{attribute 'GeneratedUsingTerminal: EP3356-0022-0016'}
{attribute addProperty BoxType "EP3356-0022-0016"}
{attribute addProperty Id "CtrlAT %Q*Ctrl_B9DDD3FF5"}
{attribute addProperty CRC "3427370076"}
{attribute addProperty Size "5"}
TYPE RMB_Control_CC49845C :
STRUCT
	{attribute addProperty Name "Ctrl"}
	Ctrl AT %Q* : Ctrl_B9DDD3FF;
END_STRUCT
END_TYPE

(* stored: Version 1.2.0.0, ProductVersion 3.1.4024.9
   DUT RMB_Control_CC49845C: Id {f68fbd6b-4ac3-407a-bedf-f95f8487c6f4} *)
